{attribute 'enable_dynamic_creation'}
FUNCTION_BLOCK PUBLIC NullEntry EXTENDS FileSystemEntry IMPLEMENTS I_NullEntry
VAR
END_VAR

PROPERTY PUBLIC IsNull : BOOL
GET
IsNull := TRUE;
END_GET
END_PROPERTY

END_FUNCTION_BLOCK

(* stored: Version 1.1.0.1, ProductVersion 3.1.4024.9
   POU NullEntry: Id {dab7c663-100f-4da6-b5ad-a2455b58ddfb}, SpecialFunc None
   Property IsNull: Id {99f7d355-bb3c-46b3-8bdf-024693cad850}
   Get Get: Id {7356c8d2-f8db-4737-ab2e-ec93d8f68b71} *)
